(* PLC project PLC, Beckhoff Automation GmbH TwinCAT PLC Control 3.5.13.21 *)
(* stored: creationDateTime 2024-02-17T22:43:12.2264758, modificationDateTime 2024-02-17T22:43:12.2264758 *)

TYPE PBInput :
STRUCT
	pushed AT %I*: BOOL;
END_STRUCT
END_TYPE
